// TIA Portal V19 export
VAR_GLOBAL   // PLC tag table "Default tag table"
   TEST_STR AT %I8.0 : Bool;
   Motor1 AT %Q8.0 : Bool;
   Stop_BTN AT %I8.1 : Bool;
END_VAR
